// TIA Portal V21 export
VAR_GLOBAL   // PLC tag table "K_Esempio"
END_VAR
VAR_GLOBAL CONSTANT   // user constants
   K_Analogica_Esempio : Int := 0;
   K_Comunicazione_Esempio : Int := 0;
   K_Motore_Esempio : Int := 0;
   K_Valvola_Esempio : Int := 0;
   K_Totalizzatore_Esempio : Int := 0;
   K_Zona_Esempio : Int := 0;
   K_SezionePastorizzatore_Esempio : Int := 0;
   K_Portata_Esempio : Int := 0;
   K_Pid_Esempio : Int := 0;
   K_Paratia_Esempio : Int := 0;
   K_Additivo_Esempio : Int := 0;
END_VAR
